{attribute 'GeneratedUsingTerminal: EL5032-0000-0021'}
{attribute addProperty BoxType "EL5032-0000-0021"}
{attribute addProperty Id "WarningBOOL1ErrorBOOL1ReadyBOOL1DiagBOOL1TxPDO_StateBOOL1Input_cycle_counterBYTE1"}
{attribute addProperty CRC "2180949863"}
{attribute addProperty Size "6"}
TYPE Status_81FEA767 :
STRUCT
	{attribute addProperty Name "Warning"}
	Warning : BOOL;
	{attribute addProperty Name "Error"}
	Error : BOOL;
	{attribute addProperty Name "Ready"}
	Ready : BOOL;
	{attribute addProperty Name "Diag"}
	Diag : BOOL;
	{attribute addProperty Name "TxPDO_State"}
	TxPDO_State : BOOL;
	{attribute addProperty Name "Input_cycle_counter"}
	Input_cycle_counter : BYTE;
END_STRUCT
END_TYPE

(* stored: Version 1.2.0.0, ProductVersion 3.1.4024.9
   DUT Status_81FEA767: Id {6b8598e9-6405-46f8-a05d-c1d6ab8259ac} *)
